// TwinCAT 3 PLC project Example
// ProgramVersion: 3.1.4024.0
// libraries:
//   MTP, * (Zerlauth)
//   Tc2_MC2, * (Beckhoff Automation GmbH)
//   Tc2_Standard, * (Beckhoff Automation GmbH)
//   Tc2_System, * (Beckhoff Automation GmbH)
//   Tc2_Utilities, * (Beckhoff Automation GmbH)
//   Tc3_Module, * (Beckhoff Automation GmbH)
// project tree:
//   / plcTask1.TcTTO
//   POUs/Axis/ FB_McAxis.TcPOU (not stored), I_Axis.TcIO (not stored)
//   POUs/ FB_Alarm.TcPOU, FB_ComponentEX.TcPOU, FB_Module01.TcPOU, MAIN.TcPOU
// real-time tasks:
//   TASK plcTask1: cycle T#25000us, priority 20, ADS port 350

CONFIGURATION Example
    RESOURCE PLC ON TwinCAT3
        TASK plcTask1(INTERVAL := T#1000ms, PRIORITY := 20);
        PROGRAM MAIN WITH plcTask1 : MAIN;
    END_RESOURCE
END_CONFIGURATION

// ---- POUs/MAIN.TcPOU
PROGRAM MAIN
VAR
	fbModule1:		FB_Module01;	
	bReset:			BOOL;
	bStart: 		BOOL;
    bHold:       	BOOL;
    bPause:    		BOOL;
	bStop:       	BOOL;
    bAbort:      	BOOL;

END_VAR


fbModule1();

IF bReset THEN
	bReset:= NOT fbModule1.M_Request(E_Request.Reset);
END_IF

IF bStart THEN
	bStart:= NOT fbModule1.M_Request(E_Request.Start);
END_IF

IF bStop THEN
	bStop:= fbModule1.M_Request(E_Request.Stop);
END_IF

IF bHold THEN
	bHold:= NOT fbModule1.M_Request(E_Request.Hold);
END_IF

IF bPause THEN
	bPause:= NOT fbModule1.M_Request(E_Request.Pause);
END_IF

IF bAbort THEN
	bAbort:= NOT fbModule1.M_Request(E_Request.Abort);
END_IF

END_PROGRAM

// ---- POUs/FB_Module01.TcPOU
FUNCTION_BLOCK FB_Module01 EXTENDS FB_Component
VAR_INPUT
	bPowerOn:				BOOL;
	bFuse1:					BOOL;
END_VAR
VAR_OUTPUT
END_VAR
VAR
	fbLogger:					FB_ListLogger;
	fbAlarm:					FB_Alarm;
	fbComponent1:				FB_Component;
	fbComponent2:				FB_Component;
	fbComponent3:				FB_Component;
	fbComponent4:				FB_ComponentEX;
	nIndex:						INT;
	fbComponent:				ARRAY[1..10000] OF FB_Component;
END_VAR

SUPER^();

fbComponent1();
fbComponent2();
fbComponent3();
fbComponent4();

FOR nIndex:= 1 TO 10000 DO 
	fbComponent[nIndex]();
END_FOR;

METHOD PROTECTED M_Initialise : BOOL
VAR_INPUT
END_VAR
IF SUPER^.M_Initialise() THEN
	fbEvent.P_Logger:= fbLogger;
	fbLogger.M_Add(fbAlarm);

	fbComponent1.fbEvent.P_Logger:= fbLogger;
	fbComponent1.fbObserver.M_Attach(THIS^);
	fbObserver.M_Attach(fbComponent1);
	
	fbComponent2.fbEvent.P_Logger:= fbLogger;
	fbComponent2.fbObserver.M_Attach(THIS^);
	fbObserver.M_Attach(fbComponent2);
	
	fbComponent3.fbEvent.P_Logger:= fbLogger;
	fbComponent3.fbObserver.M_Attach(THIS^);
	fbObserver.M_Attach(fbComponent3);
	
	fbComponent4.fbEvent.P_Logger:= fbLogger;
	fbComponent4.fbObserver.M_Attach(THIS^);
	fbObserver.M_Attach(fbComponent4);
	
	FOR nIndex:= 1 TO 10000 DO 
		fbComponent[nIndex].fbEvent.P_Logger:= fbLogger;
		fbComponent[nIndex].fbObserver.M_Attach(THIS^);
		fbObserver.M_Attach(fbComponent[nIndex]);
	END_FOR;
	
	
	
	M_Initialise:= TRUE;
END_IF
END_METHOD

METHOD PROTECTED M_Resetting : BOOL
VAR_INPUT
END_VAR
VAR
	nIndex:					DINT;
END_VAR
M_Resetting:= TRUE;
WHILE nIndex < fbObserver.nLength DO
	fbObserver.M_Index(nIndex).M_Request(E_Request.Reset);
	nIndex:= nIndex +1;
END_WHILE

fbAlarm.M_Reset();
END_METHOD

METHOD PROTECTED M_Running
VAR_INPUT
END_VAR
IF NOT bPowerOn THEN
	fbEvent.M_Add('Test');
	fbEvent.M_Add('Test2');
	fbEvent.M_Add('Test3');
	fbEvent.M_Error('Power not on', 2 ,E_Behaviour.Abort);
ELSIF NOT bFuse1 THEN
	fbEvent.M_Add('Test');
	fbEvent.M_Add('Test2');
	fbEvent.M_Add('Test3');
	fbEvent.M_Error('Fuse Triped', 3 ,E_Behaviour.Stop);	
	
END_IF
END_METHOD

METHOD PROTECTED M_Starting : BOOL
VAR_INPUT
END_VAR
VAR
	nIndex:					DINT;
END_VAR
M_Starting:= TRUE;
WHILE nIndex < fbObserver.nLength DO
	M_Starting:= M_Starting AND fbObserver.M_Index(nIndex).M_Request(E_Request.Start);
	nIndex:= nIndex +1;
END_WHILE
END_METHOD

END_FUNCTION_BLOCK

// ---- POUs/FB_Alarm.TcPOU
FUNCTION_BLOCK FB_Alarm IMPLEMENTS I_Logger
VAR_INPUT
END_VAR
VAR_OUTPUT
END_VAR
VAR
	nLength:		INT;
	aEvent:						ARRAY [0..99] OF ST_Event;
END_VAR

METHOD M_Find : DINT
VAR_INPUT
	stEvent	: 		ST_Event;
END_VAR
VAR
	nIndex: 	DINT;
END_VAR
// Object already in List
M_Find := -1;
nIndex:= 0;
WHILE nIndex < nLength DO
    IF (aEvent[nIndex].Source = stEvent.Source) 
		AND_THEN (aEvent[nIndex].EventType = stEvent.EventType) 
		AND_THEN (aEvent[nIndex].Message = stEvent.Message) THEN
			M_Find := nIndex;
			RETURN;
    END_IF
	nIndex := nIndex + 1;
END_WHILE
END_METHOD

METHOD M_Log
VAR_INPUT
	stEvent	: 		ST_Event;
END_VAR

VAR
	nIndex: DINT;
END_VAR
IF M_Find(stEvent) = -1 THEN
	aEvent[nLength]:= stEvent;
	nLength:= nLength + 1;
END_IF
END_METHOD

METHOD PUBLIC M_Reset
VAR_INPUT
END_VAR
nLength:= 0;
Tc2_System.MEMSET(adr(aEvent), 0, sizeof(aEvent));
END_METHOD

END_FUNCTION_BLOCK

// ---- POUs/FB_ComponentEX.TcPOU
FUNCTION_BLOCK FB_ComponentEX EXTENDS FB_Component
VAR_INPUT
END_VAR
VAR_OUTPUT
END_VAR
VAR
	bEvent:			BOOL;
END_VAR

SUPER^();

METHOD PROTECTED M_Execute : BOOL
VAR_INPUT
END_VAR

IF bEvent THEN
	bEvent:= FALSE;
	fbEvent.M_Add('Test');
	fbEvent.M_Add('Test2');
	fbEvent.M_Add('Test3');
	fbEvent.M_Error('First Error Abort', 1 ,E_Behaviour.Abort);
END_IF
END_METHOD

END_FUNCTION_BLOCK
